// TIA Portal V20 export
DATA_BLOCK "InstEmDataHmi"   // DB44
TITLE = Instance of FB instance of FB EnergyMeterDataToHmi
AUTHOR : SICAR
FAMILY : Energy
VERSION : 1.0
// Energy meter HMI
// stored: InstanceOfName LSicar_EnMeterDataToHmi, InstanceOfType FB
"LSicar_EnMeterDataToHmi"
   // VAR_INPUT
   //    energyMeter01Visu { ExternalAccessible := 'False'; ExternalVisible := 'False'; ExternalWritable := 'False'} : "LSicar_typeEnMeterVisuStruct";
   //    energyMeter02Visu { ExternalAccessible := 'False'; ExternalVisible := 'False'; ExternalWritable := 'False'} : "LSicar_typeEnMeterVisuStruct";
   //    energyMeter03Visu { ExternalAccessible := 'False'; ExternalVisible := 'False'; ExternalWritable := 'False'} : "LSicar_typeEnMeterVisuStruct";
   //    energyMeter04Visu { ExternalAccessible := 'False'; ExternalVisible := 'False'; ExternalWritable := 'False'} : "LSicar_typeEnMeterVisuStruct";
   //    energyMeter05Visu { ExternalAccessible := 'False'; ExternalVisible := 'False'; ExternalWritable := 'False'} : "LSicar_typeEnMeterVisuStruct";
   //    energyMeter06Visu { ExternalAccessible := 'False'; ExternalVisible := 'False'; ExternalWritable := 'False'} : "LSicar_typeEnMeterVisuStruct";
   //    energyMeter07Visu { ExternalAccessible := 'False'; ExternalVisible := 'False'; ExternalWritable := 'False'} : "LSicar_typeEnMeterVisuStruct";
   //    energyMeter08Visu { ExternalAccessible := 'False'; ExternalVisible := 'False'; ExternalWritable := 'False'} : "LSicar_typeEnMeterVisuStruct";
   // END_VAR
   // VAR
   //    statEmIndex : Int;
   //    statEmData : "LSicar_typeEnMeterVisuStruct";
   //    statResetMinMaxAll : Bool;
   //    statResetMinMax : Array[0..8] of Bool;
   //    statResetEnCounterAll : Bool;
   //    statResetEnCounter : Array[0..8] of Bool;
   // END_VAR
BEGIN
END_DATA_BLOCK
